// TIA Portal V19 export
TYPE "ValveMachine_Config"
// stored: Access Published
   STRUCT
      DelayPressureRunningTimeout : Time := T#3s;   // Ritardo attivazione warning manacanza Cin.PressureRunning
      DelayMissingCondition : Time := T#3s;   // Ritardo attivazione warning mancanza #Cin.Rest_ExtEnable / #Cin.Work_ExtEnable
      Rest_LsQty : Int;   // Numero di finecorsa REXT (multi cilindro azionati da unica valvola)
      Work_LsQty : Int;   // Numero di finecorsa WORK (multi cilindro azionati da unica valvola)
      Rest_RetainAut : Bool;   // Mantieni comando REST Aut anche dopo perdita Control_ON
      Work_RetainAut : Bool;   // Mantieni comando WORK Aut anche dopo perdita Control_ON
      V : "ValveConfig";   // configurations & parameters
   END_STRUCT;
   // V.RestLimSwitchExist := FALSE;
   // V.WorkLimSwitchExist := FALSE;
   // V.CheckOilInPressure := FALSE;
   // V.CutRestWhenIsAtRest := TRUE;
   // V.CutWorkWhenIsAtWork := TRUE;
   // V.RestTime := T#0ms;
   // V.WorkTime := T#0ms;
   // V.RestTimeOut := T#1H;
   // V.WorkTimeOut := T#1H;
END_TYPE
